(* CODESYS project lib_basic.library
   Company: Beckhoff_GZ
   Title: Lib_Basic
   Placeholder: Lib_Basic
   Version: 1.0.1.0

Project tree, tasks and I/O mapping:
  libraries: Tc2_Standard, * (Beckhoff Automation GmbH); Tc2_System, * (Beckhoff Automation GmbH)
  POUs/
    function F_TaskCycleTime [ST]
    function block FB_FreePulse [ST]
    function block FB_TriggerOnOff [ST]
*)

// POUs/F_TaskCycleTime
FUNCTION F_TaskCycleTime : REAL			(*获取当前 Task 周期时间, 单位: ms*)
VAR_INPUT
END_VAR
VAR
	s_fbGetCurTaskIndex	: GETCURTASKINDEX;
	s_fCurTaskTime		: REAL;
END_VAR

;
s_fbGetCurTaskIndex();
F_TaskCycleTime := TwinCAT_SystemInfoVarList._TaskInfo[s_fbGetCurTaskIndex.index].cycleTime / 1E4;		(* ms *)

END_FUNCTION

// POUs/FB_FreePulse
FUNCTION_BLOCK FB_FreePulse
VAR_INPUT
	bEnable					: BOOL	:= FALSE;	(*开始*)
	tCycleTime				: TIME	:= T#1S;	(*周期时间*)
	nDutyCycle				: UINT	:= 50;		(*脉冲输出占空比, 0-100*)
END_VAR
VAR_OUTPUT
	bOutput					: BOOL;
END_VAR
VAR
	TON1, TON2				: TON;
END_VAR

;
IF NOT bEnable THEN
	nDutyCycle := LIMIT(0, nDutyCycle, 100);
	TON1.PT := tCycleTime * (100 - nDutyCycle) / 100;	
	TON2.PT := tCycleTime * (nDutyCycle) / 100;
END_IF

IF TON2.Q THEN
	TON2.PT := tCycleTime * (nDutyCycle) / 100;
END_IF

TON1(IN := bEnable);
TON2(IN := TON1.Q);

IF TON2.Q THEN
	nDutyCycle := LIMIT(0, nDutyCycle, 100);	
	TON1(IN := FALSE);
	TON1(IN := bEnable, PT := tCycleTime * (100 - nDutyCycle) / 100);
END_IF

bOutput := TON1.Q;

END_FUNCTION_BLOCK

// POUs/FB_TriggerOnOff
FUNCTION_BLOCK FB_TriggerOnOff		(*单按钮控制输出, 状态取反*)
VAR_INPUT
	bTrigger				: BOOL	:= FALSE;		(*按钮输入*)
	bSetOff					: BOOL	:= TRUE;		(*强制复位输出*)
END_VAR
VAR_OUTPUT
END_VAR
VAR_IN_OUT
	bOnOff					: BOOL;					(*输出, 可在外部程序复位该变量*)
END_VAR
VAR
	s_rtTrigger				: R_TRIG;
END_VAR

;
s_rtTrigger(CLK := bTrigger);
IF bSetOff THEN
	bOnOff := FALSE;
ELSE
	IF s_rtTrigger.Q THEN
		bOnOff := NOT bOnOff;
	END_IF
END_IF

END_FUNCTION_BLOCK
